// TwinCAT 3 PLC project Untitled1
// ProgramVersion: 3.1.4022.7
// libraries:
//   Tc2_Standard, * (Beckhoff Automation GmbH)
//   Tc2_System, * (Beckhoff Automation GmbH)
//   Tc3_Module, * (Beckhoff Automation GmbH)
//   VisuDialogs, * (System)
//   VisuSymbols,3.5.10.0,System
// project tree:
//   DUTs/ ePiston.TcDUT
//   / GlobalTextList.TcGTLO, PlcTask.TcTTO, Visualization Manager.TcVMO (not stored), VISU_TASK.TcTTO
//   POUs/ MAIN.TcPOU, Piston.TcPOU
//   VISUs/ Visualization.TcVIS, V_piston.TcVIS
// real-time tasks:
//   TASK PlcTask: cycle T#10ms, priority 20, ADS port 350
//   TASK VISU_TASK: cycle T#200000us, priority 30, ADS port 351

CONFIGURATION Untitled1
    RESOURCE PLC ON TwinCAT3
        TASK PlcTask(INTERVAL := T#10ms, PRIORITY := 20);
        TASK VISU_TASK(INTERVAL := T#200000us, PRIORITY := 30);
        PROGRAM MAIN WITH PlcTask : MAIN;
        PROGRAM VisuElems_Visu_Prg WITH VISU_TASK : VisuElems.Visu_Prg;
    END_RESOURCE
END_CONFIGURATION

// ---- DUTs/ePiston.TcDUT
{attribute 'qualified_only'}
{attribute 'strict'}
TYPE ePiston :
(
	off := 0,
	running,
	fwd,
	bkw,
	error
);
END_TYPE

// ---- POUs/MAIN.TcPOU
PROGRAM MAIN
VAR
	p1	: Piston;
	pSensor: BOOL;
	nSensor: BOOL;
	pOut: BOOL;
	nOut: BOOL;
	timeOut: TIME := T#5S;
	delay: TIME := T#2S;
	noSensorTimeout: TIME := T#2S;
	pbSetTimers: BOOL;
END_VAR


p1(
	pSensor:= pSensor , 
	nSensor:= nSensor, 
	pistonName:= 'Test Piston' , 
	pOut=> pOut, 
	nOut=> nOut, 
	error=> , 
	isBusy=> , 
	errormessage=> , 
	sState=> , 
	isBKW=> , 
	isFWD=> , 
	isOFF=> );
	
IF pbSetTimers THEN
	p1.setTimers(T#5S, T#5S, T#5S);
END_IF

END_PROGRAM

// ---- POUs/Piston.TcPOU
FUNCTION_BLOCK Piston
VAR_INPUT
	pSensor, nSensor : BOOL;
	pistonName : STRING;
END_VAR
VAR_OUTPUT
	pOut, nOut, error, isBusy : BOOL;
	errormessage: STRING(255);
	sState: STRING; // state of the piston
	isBKW: BOOL;
	isFWD: BOOL;
	isOFF: BOOL;
END_VAR
VAR
	_timeOut : TIME:= T#5S; // running the task timeout
	_delay : TIME:= T#1S; // in position (on sensor) timeout
	_noSensorTimeout : TIME:= T#2S; // sensor lost in FWD or BKW state
	timeOutTimer, delayTimer, noSensorTimeoutTimer : ton;
	state,task : ePiston;
	execute: BOOL; // run method with task input
	trExecute: R_trig;
	// testing rise error
	testError: BOOL; 
	//STEP mode - no use in this FB
	nextStep: BOOL;
	stepMode: BOOL;
	stepPB: BOOL;
	trStepPB: R_trig;
	sTask: STRING;
END_VAR

delayTimer(IN:= state=ePiston.running AND 
				(((task=ePiston.bkw) AND nSensor) OR
				((task=ePiston.fwd) AND pSensor)),
 		   PT:=_delay);
////////////////////////////////////////////////////////////////
timeOutTimer(IN:= state=ePiston.running AND
				  (((task=ePiston.bkw) AND NOT nSensor) OR 
				  ((task=ePiston.fwd) AND NOT pSensor)),
			 PT:=_timeOut);
////////////////////////////////////////////////////////////////
noSensorTimeoutTimer(IN:= (state=ePiston.fwd AND NOT pSensor) OR 
						  (state=episton.bkw AND NOT nSensor),
			 		 PT:= _noSensorTimeout );
////////////////////////////////////////////////////////////////
CASE state OF
	ePiston.off: // wait for execute trigger
		M_off();
	ePiston.running:
		IF M_run() THEN
			execute := FALSE;
			M_SetState(task);
		END_IF
	ePiston.fwd: // wait for execute trigger
		M_fwd();
	ePiston.bkw: // wait for execute trigger
		M_bkw();
	ePiston.error: // wait for reset method (from outside)
		M_off();
END_CASE
///////////////////////////////////////////////////////////////////////
statesIndication();
///////////////////////////////////////////////////////////////////////
trExecute(clk:=execute);
IF trExecute.Q AND state<>ePiston.error AND state<>ePiston.running THEN
			M_SetState(ePiston.running);
END_IF
///////////////////////////////////////////////////////////////////////
IF pSensor AND nSensor THEN
	M_riseError('- 2 sensors in one time - not acceptable!');
END_IF
///////////////////////////////////////////////////////////////////////
IF NOT error AND testError THEN // testing
	M_riseError('- testing error');
END_IF
///////////////////////////////////////////////////////////////////////
// STEP MODE
stepMode := FALSE; // STEP MODE not used
trStepPB(CLK:=stepPB);
nextStep := NOT stepMode OR trStepPB.Q; // for the M_SetState method  
///////////////////////////////////////////////////////////////////////

METHOD PUBLIC bkw : BOOL
VAR_INPUT
END_VAR
IF NOT execute AND state<>ePiston.error AND state<>ePiston.running
	AND state<>ePiston.bkw
	 THEN
	task := ePiston.bkw;
	execute := TRUE;
END_IF
END_METHOD

METHOD PUBLIC fwd : BOOL
VAR_INPUT
END_VAR
IF NOT execute AND state<>ePiston.error AND state<>ePiston.running
	AND state<>ePiston.fwd
	 THEN
	task := ePiston.fwd;
	execute := TRUE;
END_IF
END_METHOD

METHOD PRIVATE M_bkw : BOOL
VAR_INPUT
END_VAR
VAR
	//bkwState : BOOL;
END_VAR
pout := FALSE;
nout := TRUE;

IF state=ePiston.bkw AND (noSensorTimeoutTimer.Q OR pSensor) THEN
	M_riseError('- error in BKW - check the sensor');
END_IF
END_METHOD

METHOD PRIVATE M_fwd : BOOL
VAR_INPUT
END_VAR
VAR
	//fwdState : BOOL;
END_VAR
pout := TRUE;
nout := FALSE;

IF state=ePiston.fwd AND (noSensorTimeoutTimer.Q OR nSensor) THEN
	M_riseError('- error in FWD - check the sensor');
END_IF
END_METHOD

METHOD PRIVATE M_off : BOOL
VAR_INPUT
END_VAR
pOut := FALSE;
nOut := FALSE;
END_METHOD

METHOD PRIVATE M_riseError : BOOL
VAR_INPUT
	message : STRING;
END_VAR
errormessage := CONCAT(pistonName, message);

IF NOT error THEN
	error := TRUE;
	M_SetState(episton.error);
	//TODO log with message
END_IF
END_METHOD

METHOD PRIVATE M_run : BOOL
VAR_INPUT
	//task : INT; // enum
END_VAR
CASE task OF
	ePiston.off:
		M_off();
		M_run := TRUE;
	ePiston.bkw:
		M_bkw();
	ePiston.fwd:
		M_fwd();
END_CASE
sTask := stateToString(task);

IF delayTimer.Q THEN
	sTask := '';
	M_run := TRUE;
ELSIF timeOutTimer.Q THEN
	M_riseError(CONCAT('- timeout in the task: ' , stateToString(task)));
END_IF
END_METHOD

METHOD PRIVATE M_SetState
VAR_INPUT
	eNextState : ePiston; //INT;
END_VAR
IF State <> eNextState AND nextStep THEN
	//AddEventToLog(State,SeverityLevelType.Info,f_concat9( 'Changing State FROM ', M_statetostring(State), 'TO' ,M_StateToString(eNextState),'','','','',''));
	State := eNextState;
	//stateString := M_statetostring(State);
END_IF
END_METHOD

METHOD PUBLIC off : BOOL
VAR_INPUT
END_VAR
IF NOT execute AND state<>ePiston.error AND state<>ePiston.running 
	AND state<>ePiston.off
	THEN
	task := ePiston.off;
	execute := TRUE;
END_IF
END_METHOD

METHOD reset : BOOL
VAR_INPUT
END_VAR
IF state = episton.error OR error THEN
	M_SetState(ePiston.off);
	execute := FALSE;
	error := FALSE;
	errormessage := '';
END_IF
END_METHOD

METHOD PUBLIC setTimers : BOOL
VAR_INPUT
	timeOut : TIME; // running the task timeout
	delay : TIME; // in position (on sensor) timeout
	noSensorTimeout : TIME; // sensor lost in FWD or BKW state
END_VAR
_timeOut			:= timeOut;
_delay				:= delay;
_noSensorTimeout	:= noSensorTimeout;
END_METHOD

ACTION statesIndication:
isBKW := state = ePiston.bkw;
isFWD := state = ePiston.fwd;
isOFF := state = ePiston.off;
isBusy := state = ePiston.running;

sState := stateToString(state);
END_ACTION

METHOD PRIVATE stateToString : string
VAR_INPUT
	ePistonState : INT; // ePiston enum
END_VAR
CASE ePistonState OF
	ePiston.bkw:
		stateToString := 'BKW';
	ePiston.fwd:
		stateToString := 'FWD';
	ePiston.error:
		stateToString := 'ERROR';
	ePiston.off:
		stateToString := 'OFF';
	ePiston.running:
		stateToString :=concat('RUNNING ', sTask);
END_CASE
END_METHOD

END_FUNCTION_BLOCK

// ---- GlobalTextList.TcGTLO
TEXTLIST GlobalTextList
  997 = '%s'
  992 = 'BKW'
  916 = 'delay'
  829 = 'FWD'
  203 = 'noSensorTimeout'
  843 = 'nOUT'
  331 = 'nSensor'
  871 = 'OFF'
  406 = 'PB set timers'
  609 = 'pOUT'
  306 = 'pSensor'
  970 = 'Reset'
  70 = 'timeOut'
END_TEXTLIST

// ---- VISUs/Visualization.TcVIS
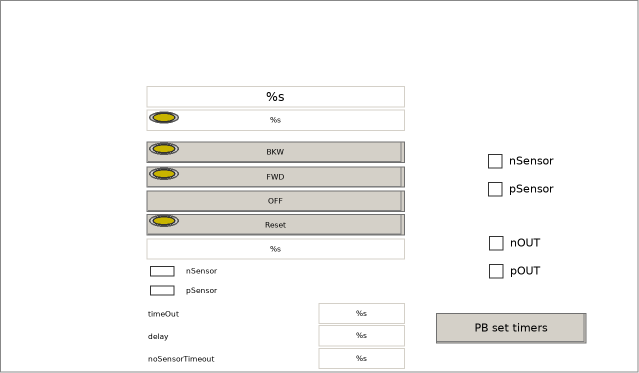
VISUALIZATION Visualization  // 639x373
    Frame (121,78 287x293)
        shows V_piston(p := MAIN.p1)
    Checkbox (486,146 150x30), "nSensor", variable: MAIN.nSensor
    Checkbox (486,174 150x30), "pSensor", variable: MAIN.pSensor
    Checkbox (487,228 150x30), "nOUT", variable: MAIN.nOut
    Checkbox (487,256 150x30), "pOUT", variable: MAIN.pOut
    Button (436,313 150x30), "PB set timers"
        OnMouseClick: toggle MAIN.pbSetTimers
END_VISUALIZATION

// ---- VISUs/V_piston.TcVIS
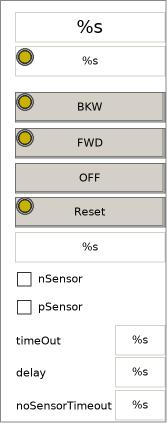
VISUALIZATION V_piston  // 167x423
VAR_IN_OUT
	p : piston;
END_VAR
    Textfield (15,12 150x30), "%s", text variable: p.pistonName
    Button (15,128 150x30), "FWD"
        OnMouseClick: execute { P.fwd(); }
    Textfield (15,46 150x30), "%s", text variable: p.sState
    Button (15,92 150x30), "BKW"
        OnMouseClick: execute { P.bkw(); }
    Button (15,163 150x30), "OFF"
        OnMouseClick: execute { P.off(); }
    Button (15,197 150x30), "Reset"
        OnMouseClick: execute { P.reset(); }
    Lamp1 (15,196 20x20), variable: p.error, style: Lamp-Lamp1-Yellow
    Lamp1 (15,47 20x20), variable: p.isBusy, style: Lamp-Lamp1-Yellow
    Textfield (15,232 150x30), "%s", text variable: p.errormessage
    Checkbox (15,264 150x30), "nSensor", variable: p.nSensor
    Checkbox (15,292 150x30), "pSensor", variable: p.pSensor
    Lamp1 (15,92 20x20), variable: p.nOut, style: Lamp-Lamp1-Yellow
    Lamp1 (15,128 20x20), variable: p.pOut, style: Lamp-Lamp1-Yellow
    Textfield (115,325 50x30), "%s", text variable: p._timeOut
        OnMouseClick: write the text variable via Default
    Label (13,326 110x30), "timeOut"
    Textfield (115,357 50x30), "%s", text variable: p._delay
        OnMouseClick: write the text variable via Default
    Label (13,358 110x30), "delay"
    Textfield (115,390 50x30), "%s", text variable: p._noSensorTimeout
        OnMouseClick: write the text variable via Default
    Label (13,391 110x30), "noSensorTimeout"
END_VISUALIZATION
